// TIA Portal V20 export
DATA_BLOCK "DemoLoopInstance"   // DB40
// stored: InstanceOfName DemoLoopFB, InstanceOfType FB
"DemoLoopFB"
   // VAR_IN_OUT
   //    Loop : DemoController;
   //    Link : "DemoUdt";
   // END_VAR
   // VAR RETAIN
   //    Settings { S7_SetPoint := 'True'} : "DemoSettings";
   // END_VAR
BEGIN
   Settings.Limits.Upper := 30.0;
   Settings.Limits.Lower := 9.0;
   Settings.Mode := 1;
END_DATA_BLOCK
